(*			
	RafalOS
	Rafał Osajda		10.11.2025		TC 4024.66
	Główny blok konfiguracyjny MachineControl
*)
FUNCTION_BLOCK FB_MachineDefaultConfiguration EXTENDS FB_Base IMPLEMENTS ITF_MCConfiguration
VAR

END_VAR

METHOD PUBLIC AddHMIToMachineControl : BOOL
VAR_INPUT
	itfMachineControl			: ITF_MCMachineControlConfigure;
END_VAR
itfMachineControl.AddHMIManager (itfHMIManager := GVL_SystemVariable.fbHMIManager);
END_METHOD

METHOD PUBLIC AddTopElementToLogger : BOOL
VAR_INPUT
END_VAR
GVL_SystemVariable.fbMachineControl.JoinTheLogger ();
END_METHOD

(*			
	RafalOS
	Rafał Osajda		29.10.2025		TC 4024.66
	Dodawanie TopElementu do systemu
*)
METHOD PUBLIC AddTopElementToMachineControl : BOOL
VAR_INPUT
	itfMachineControl			: ITF_MCMachineControlConfigure;
END_VAR
THIS^.SetText (eLocation := E_BaseLocation.pl, wsDescription := "System");
THIS^.SetText (eLocation := E_BaseLocation.en, wsDescription := "System");
THIS^.SetText (eLocation := E_BaseLocation.de, wsDescription := "System");
GVL_SystemVariable.fbMachineControl.SetName (stName := THIS^.GetTexts ());
itfMachineControl.AddTopElementFromConfiguration (fbTopElement	:= GVL_SystemVariable.fbMachineControl);
END_METHOD

METHOD PUBLIC SetStartMode : BOOL
VAR_INPUT
	itfMachineControl			: ITF_MCMachineControlConfigure;
END_VAR
itfMachineControl.SetStartMode (eStartMode := E_BaseMachineMode.Production);
END_METHOD

METHOD StateAndModes : BOOL
VAR_INPUT
	itfMachineControl			: ITF_MCMachineControlConfigure;
END_VAR
itfMachineControl.AddRequestStateChange (iNumberOfRequest := E_SaMCommandChangeState.Clear,		itfRequest := GVL_RequeestChange.fbprClear);
itfMachineControl.AddRequestStateChange (iNumberOfRequest := E_SaMCommandChangeState.Reset, 	itfRequest := GVL_RequeestChange.fbprReset);
itfMachineControl.AddRequestStateChange (iNumberOfRequest := E_SaMCommandChangeState.Start, 	itfRequest := GVL_RequeestChange.fbprStart);
itfMachineControl.AddRequestStateChange (iNumberOfRequest := E_SaMCommandChangeState.Stop, 		itfRequest := GVL_RequeestChange.fbprStop);
itfMachineControl.AddRequestStateChange (iNumberOfRequest := E_SaMCommandChangeState.Suspend, 	itfRequest := GVL_RequeestChange.fbprSuspend);
itfMachineControl.AddRequestStateChange (iNumberOfRequest := E_SaMCommandChangeState.Unsuspend, itfRequest := GVL_RequeestChange.fbprUnsuspend);
itfMachineControl.AddRequestStateChange (iNumberOfRequest := E_SaMCommandChangeState.Hold, 		itfRequest := GVL_RequeestChange.fbprHold);
itfMachineControl.AddRequestStateChange (iNumberOfRequest := E_SaMCommandChangeState.Unhold, 	itfRequest := GVL_RequeestChange.fbprUnhold);
itfMachineControl.AddRequestStateChange (iNumberOfRequest := E_SaMCommandChangeState.Complete, 	itfRequest := GVL_RequeestChange.fbprComplete);
itfMachineControl.AddRequestStateChange (iNumberOfRequest := E_SaMCommandChangeState.Abort,		itfRequest := GVL_RequeestChange.fbprAbort);

itfMachineControl.AddRequestModeChange (iNumberOfRequest := E_SaMCommandChangeMode.Production, 	itfRequest := GVL_RequeestChange.fbprProduction);
itfMachineControl.AddRequestModeChange (iNumberOfRequest := E_SaMCommandChangeMode.Maintenance,	itfRequest := GVL_RequeestChange.fbprMaintenance);
itfMachineControl.AddRequestModeChange (iNumberOfRequest := E_SaMCommandChangeMode.Manual, 		itfRequest := GVL_RequeestChange.fbprManual);
itfMachineControl.AddRequestModeChange (iNumberOfRequest := E_SaMCommandChangeMode.Washing,		itfRequest := GVL_RequeestChange.fbprWashing);
itfMachineControl.AddRequestModeChange (iNumberOfRequest := E_SaMCommandChangeMode.Diagnostisc,	itfRequest := GVL_RequeestChange.fbprDiagnostics);
END_METHOD

END_FUNCTION_BLOCK

(* stored: Version 1.1.0.1
   POU FB_MachineDefaultConfiguration: Id {b648aa86-a7e1-098c-12e9-4759598ffa68}, SpecialFunc None
   Method AddHMIToMachineControl: Id {1ddb6eb9-c931-0e11-33e1-e42c75396327}
   Method AddTopElementToLogger: Id {332b5b16-6a8b-4f9c-b147-743d36983c25}
   Method AddTopElementToMachineControl: Id {58e1fa28-d374-49d5-b4f2-6555dd78af83}
   Method SetStartMode: Id {281bfd3c-5022-467b-b076-37f9b0db67bc}
   Method StateAndModes: Id {017f3a1b-6dcb-4e00-82fc-a658d05da483} *)
